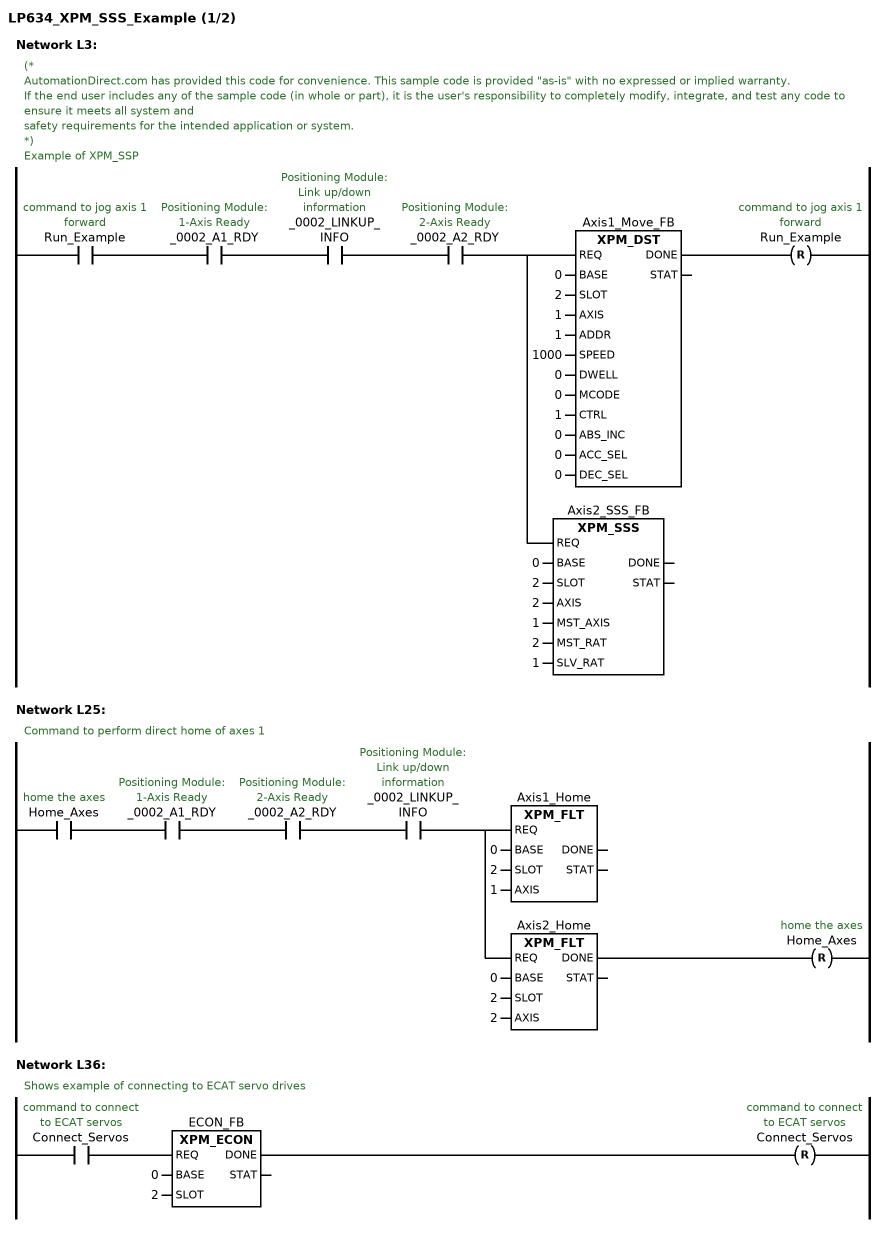
(* [picture p48: LP634_XPM_SSS_Example rungs L3-L36] *)
(* ( * / AutomationDirect.com has provided this code for convenience. This sample code is provided "as-is" with no expressed or implied warranty. / If the end user includes any of the sample code (in whole or part), it is the user's responsibility to completely modify, integrate, and test any code to ensure it meets all system and / safety requirements for the intended application or system. / * ) *)
(* Example of XPM_SSP *)
(* Rung L3 *)
_p1 := Run_Example AND _0002_A1_RDY AND _0002_LINKUP_INFO AND _0002_A2_RDY;
Axis1_Move_FB(REQ := _p1, BASE := 0, SLOT := 2, AXIS := 1, ADDR := 1, SPEED := 1000, DWELL := 0, MCODE := 0, CTRL := 1, ABS_INC := 0, ACC_SEL := 0, DEC_SEL := 0);
IF Axis1_Move_FB.DONE THEN Run_Example := FALSE; END_IF;
Axis2_SSS_FB(REQ := _p1, BASE := 0, SLOT := 2, AXIS := 2, MST_AXIS := 1, MST_RAT := 2, SLV_RAT := 1);
(* Command to perform direct home of axes 1 *)
(* Rung L25 *)
_p2 := Home_Axes AND _0002_A1_RDY AND _0002_A2_RDY AND _0002_LINKUP_INFO;
Axis1_Home(REQ := _p2, BASE := 0, SLOT := 2, AXIS := 1);
Axis2_Home(REQ := _p2, BASE := 0, SLOT := 2, AXIS := 2);
IF Axis2_Home.DONE THEN Home_Axes := FALSE; END_IF;
(* Shows example of connecting to ECAT servo drives *)
(* Rung L36 *)
ECON_FB(REQ := Connect_Servos, BASE := 0, SLOT := 2);
IF ECON_FB.DONE THEN Connect_Servos := FALSE; END_IF;

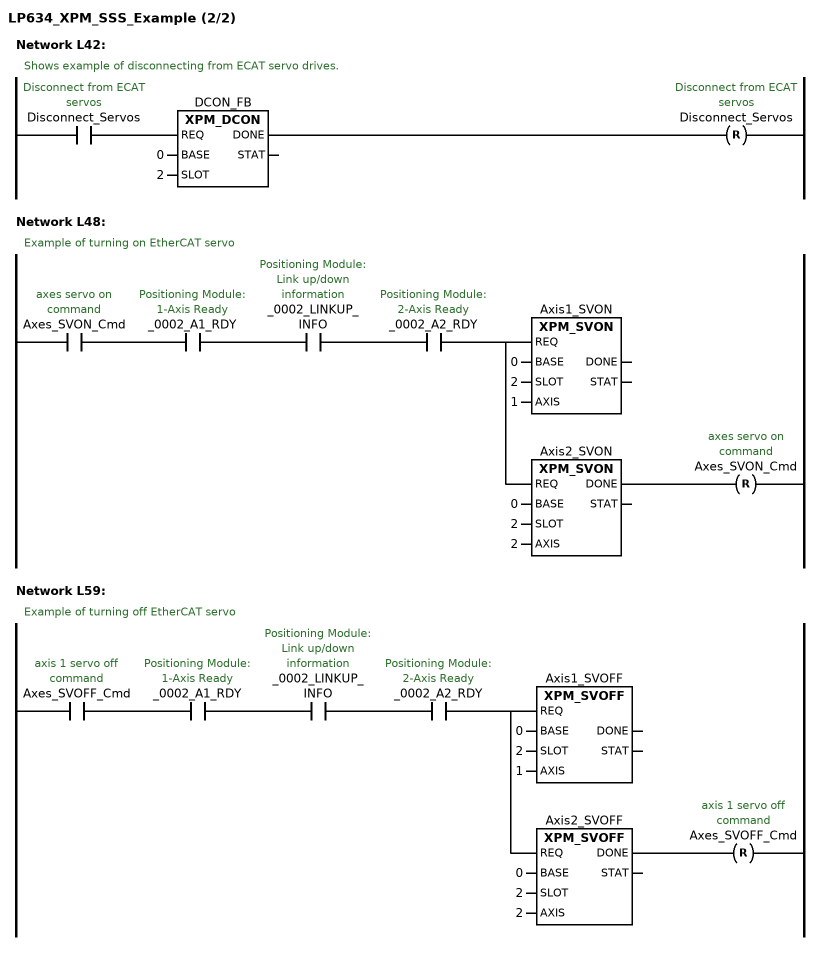
(* Shows example of disconnecting from ECAT servo drives. *)
(* Rung L42 *)
DCON_FB(REQ := Disconnect_Servos, BASE := 0, SLOT := 2);
IF DCON_FB.DONE THEN Disconnect_Servos := FALSE; END_IF;
(* Example of turning on EtherCAT servo *)
(* Rung L48 *)
_p3 := Axes_SVON_Cmd AND _0002_A1_RDY AND _0002_LINKUP_INFO AND _0002_A2_RDY;
Axis1_SVON(REQ := _p3, BASE := 0, SLOT := 2, AXIS := 1);
Axis2_SVON(REQ := _p3, BASE := 0, SLOT := 2, AXIS := 2);
IF Axis2_SVON.DONE THEN Axes_SVON_Cmd := FALSE; END_IF;
(* Example of turning off EtherCAT servo *)
(* Rung L59 *)
_p4 := Axes_SVOFF_Cmd AND _0002_A1_RDY AND _0002_LINKUP_INFO AND _0002_A2_RDY;
Axis1_SVOFF(REQ := _p4, BASE := 0, SLOT := 2, AXIS := 1);
Axis2_SVOFF(REQ := _p4, BASE := 0, SLOT := 2, AXIS := 2);
IF Axis2_SVOFF.DONE THEN Axes_SVOFF_Cmd := FALSE; END_IF;
END_PROGRAM

PROGRAM LP634_XPM_SSSP_Example (* task: Scan Program *)
(* example program for XPM_SSSP *)
VAR
    Axes_SVOFF_Cmd : BOOL; (* axis 1 servo off command *)
    Axes_SVON_Cmd : BOOL; (* axes servo on command *)
    Axis1_Home : XPM_FLT; (* direct home of axis 1 *)
    Axis1_Move_FB : XPM_DST; (* axis 1 speed move fb *)
    Axis1_SVOFF : XPM_SVOFF; (* function block for axis 1 servo off *)
    Axis1_SVON : XPM_SVON; (* SVON fb for axis 1 *)
    Axis2_Home : XPM_FLT; (* direct home of axis 1 *)
    Axis2_SSSP_FB : XPM_SSSP; (* axis 2 XPM_SSSP fb *)
    Axis2_SVOFF : XPM_SVOFF; (* function block for axis 1 servo off *)
    Axis2_SVON : XPM_SVON; (* SVON fb for axis 1 *)
    Connect_Servos : BOOL; (* command to connect to ECAT servos *)
    DCON_FB : XPM_DCON; (* EtherCAT disconnect FB *)
    Disconnect_Servos : BOOL; (* Disconnect from ECAT servos *)
    ECON_FB : XPM_ECON; (* EtherCAT connect FB *)
    Home_Axes : BOOL; (* home the axes *)
    Run_Example : BOOL; (* command to jog axis 1 forward *)
END_VAR
VAR_EXTERNAL
    _0002_A1_RDY : BOOL; (* AT %UX0.2.0 *) (* Positioning Module: 1-Axis Ready *)
    _0002_A2_RDY : BOOL; (* AT %UX0.2.1 *) (* Positioning Module: 2-Axis Ready *)
    _0002_LINKUP_INFO : BOOL; (* AT %UX0.2.14 *) (* Positioning Module: Link up/down information *)
END_VAR
VAR
    _p1 : BOOL;
    _p2 : BOOL;
    _p3 : BOOL;
    _p4 : BOOL;
END_VAR

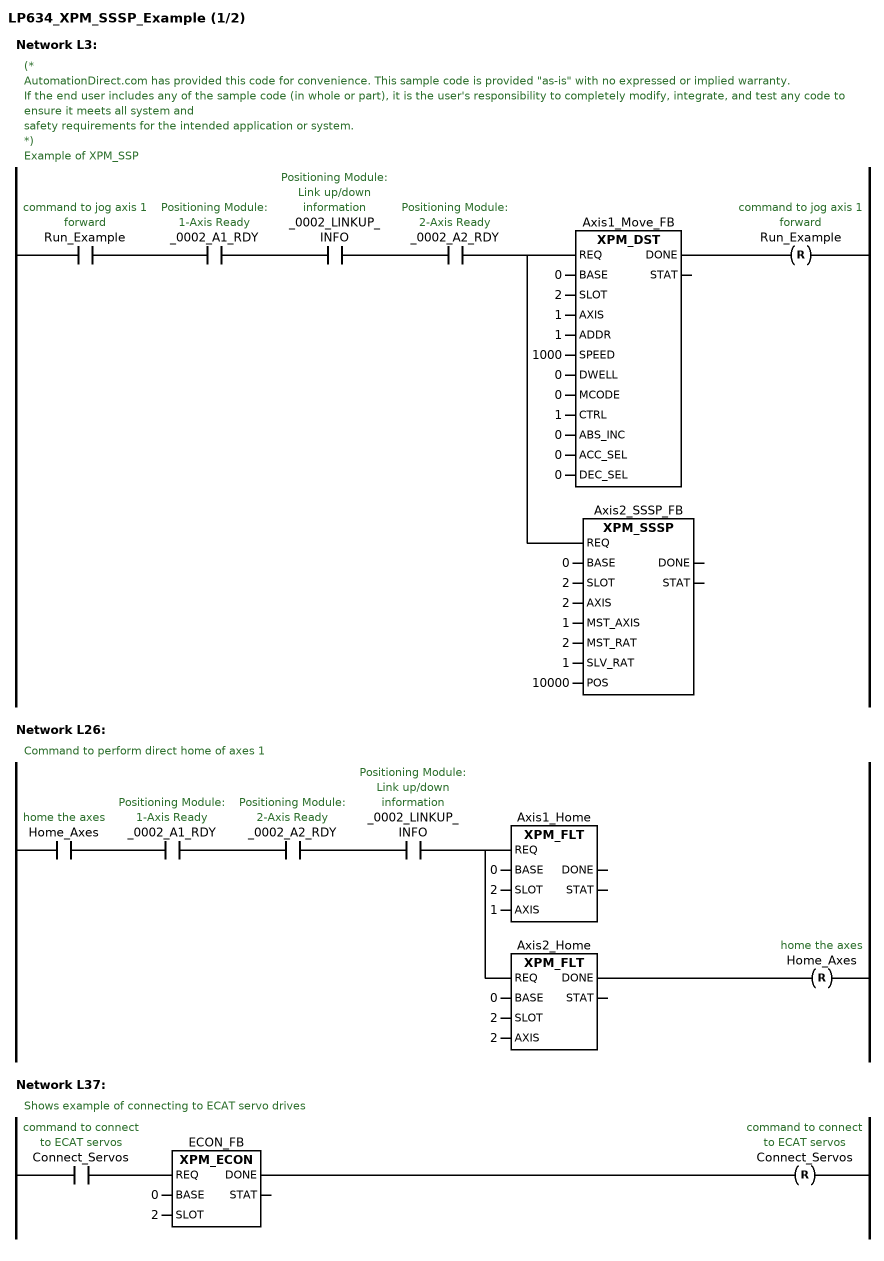
(* ( * / AutomationDirect.com has provided this code for convenience. This sample code is provided "as-is" with no expressed or implied warranty. / If the end user includes any of the sample code (in whole or part), it is the user's responsibility to completely modify, integrate, and test any code to ensure it meets all system and / safety requirements for the intended application or system. / * ) *)
(* Example of XPM_SSP *)
(* Rung L3 *)
_p1 := Run_Example AND _0002_A1_RDY AND _0002_LINKUP_INFO AND _0002_A2_RDY;
Axis1_Move_FB(REQ := _p1, BASE := 0, SLOT := 2, AXIS := 1, ADDR := 1, SPEED := 1000, DWELL := 0, MCODE := 0, CTRL := 1, ABS_INC := 0, ACC_SEL := 0, DEC_SEL := 0);
IF Axis1_Move_FB.DONE THEN Run_Example := FALSE; END_IF;
Axis2_SSSP_FB(REQ := _p1, BASE := 0, SLOT := 2, AXIS := 2, MST_AXIS := 1, MST_RAT := 2, SLV_RAT := 1, POS := 10000);
(* Command to perform direct home of axes 1 *)
(* Rung L26 *)
_p2 := Home_Axes AND _0002_A1_RDY AND _0002_A2_RDY AND _0002_LINKUP_INFO;
Axis1_Home(REQ := _p2, BASE := 0, SLOT := 2, AXIS := 1);
Axis2_Home(REQ := _p2, BASE := 0, SLOT := 2, AXIS := 2);
IF Axis2_Home.DONE THEN Home_Axes := FALSE; END_IF;
(* Shows example of connecting to ECAT servo drives *)
(* Rung L37 *)
ECON_FB(REQ := Connect_Servos, BASE := 0, SLOT := 2);
IF ECON_FB.DONE THEN Connect_Servos := FALSE; END_IF;

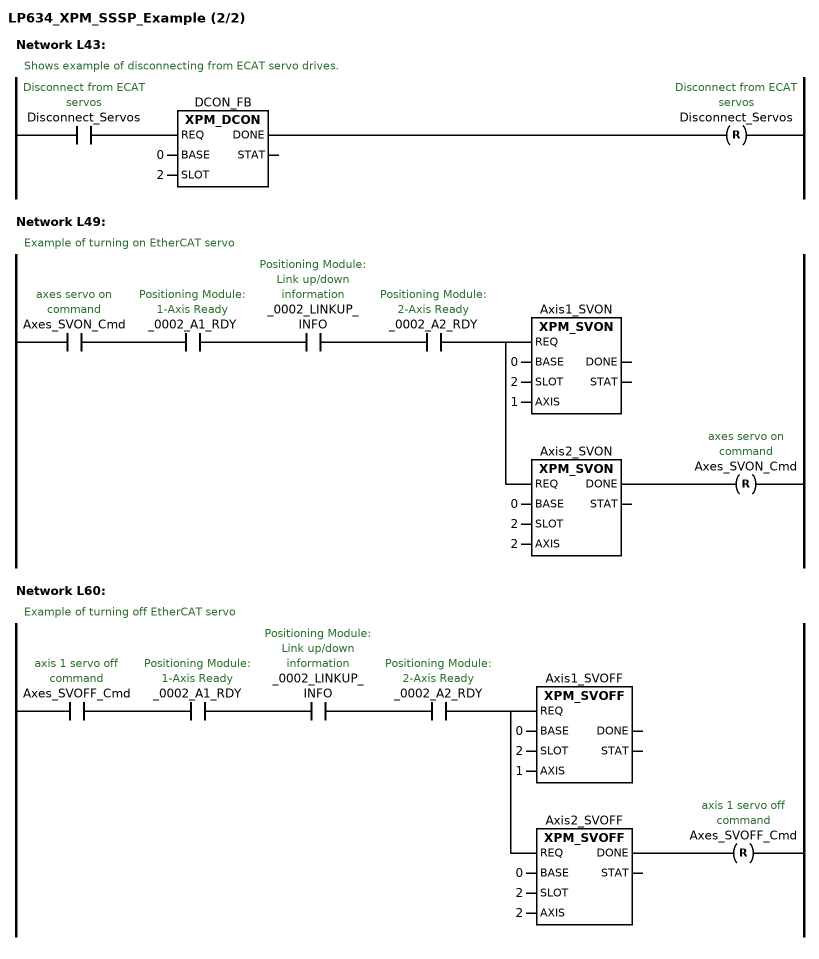
(* Shows example of disconnecting from ECAT servo drives. *)
(* Rung L43 *)
DCON_FB(REQ := Disconnect_Servos, BASE := 0, SLOT := 2);
IF DCON_FB.DONE THEN Disconnect_Servos := FALSE; END_IF;
(* Example of turning on EtherCAT servo *)
(* Rung L49 *)
_p3 := Axes_SVON_Cmd AND _0002_A1_RDY AND _0002_LINKUP_INFO AND _0002_A2_RDY;
Axis1_SVON(REQ := _p3, BASE := 0, SLOT := 2, AXIS := 1);
Axis2_SVON(REQ := _p3, BASE := 0, SLOT := 2, AXIS := 2);
IF Axis2_SVON.DONE THEN Axes_SVON_Cmd := FALSE; END_IF;
(* Example of turning off EtherCAT servo *)
(* Rung L60 *)
_p4 := Axes_SVOFF_Cmd AND _0002_A1_RDY AND _0002_LINKUP_INFO AND _0002_A2_RDY;
Axis1_SVOFF(REQ := _p4, BASE := 0, SLOT := 2, AXIS := 1);
Axis2_SVOFF(REQ := _p4, BASE := 0, SLOT := 2, AXIS := 2);
IF Axis2_SVOFF.DONE THEN Axes_SVOFF_Cmd := FALSE; END_IF;
END_PROGRAM

PROGRAM LP635_XPM_ELIN_Example (* task: Scan Program *)
(* example program for XPM_ELIN  function block. *)
VAR
    Axes_SVOFF_Cmd : BOOL; (* axis 1 servo off command *)
    Axes_SVON_Cmd : BOOL; (* axes servo on command *)
    Axis1_CMD_Step : UINT; (* step to run in XPM_IST *)
    Axis1_ELIN : XPM_ELIN; (* xpm ELIN fb *)
    Axis1_ELIN_CMD : BOOL; (* command to jog axis 1 forward *)
    Axis1_Home : XPM_FLT; (* direct home of axis 1 *)
    Axis1_SVOFF : XPM_SVOFF; (* function block for axis 1 servo off *)
    Axis1_SVON : XPM_SVON; (* SVON fb for axis 1 *)
    Axis2_Home : XPM_FLT; (* direct home of axis 1 *)
    Axis2_SVOFF : XPM_SVOFF; (* function block for axis 1 servo off *)
    Axis2_SVON : XPM_SVON; (* SVON fb for axis 1 *)
    Connect_Servos : BOOL; (* command to connect to ECAT servos *)
    DCON_FB : XPM_DCON; (* EtherCAT disconnect FB *)
    Disconnect_Servos : BOOL; (* Disconnect from ECAT servos *)
    ECON_FB : XPM_ECON; (* EtherCAT connect FB *)
    Home_Axes : BOOL; (* home the axes *)
END_VAR
VAR_EXTERNAL
    _0002_A1_RDY : BOOL; (* AT %UX0.2.0 *) (* Positioning Module: 1-Axis Ready *)
    _0002_A2_RDY : BOOL; (* AT %UX0.2.1 *) (* Positioning Module: 2-Axis Ready *)
    _0002_LINKUP_INFO : BOOL; (* AT %UX0.2.14 *) (* Positioning Module: Link up/down information *)
END_VAR
VAR
    _p1 : BOOL;
    _p2 : BOOL;
    _p3 : BOOL;
END_VAR

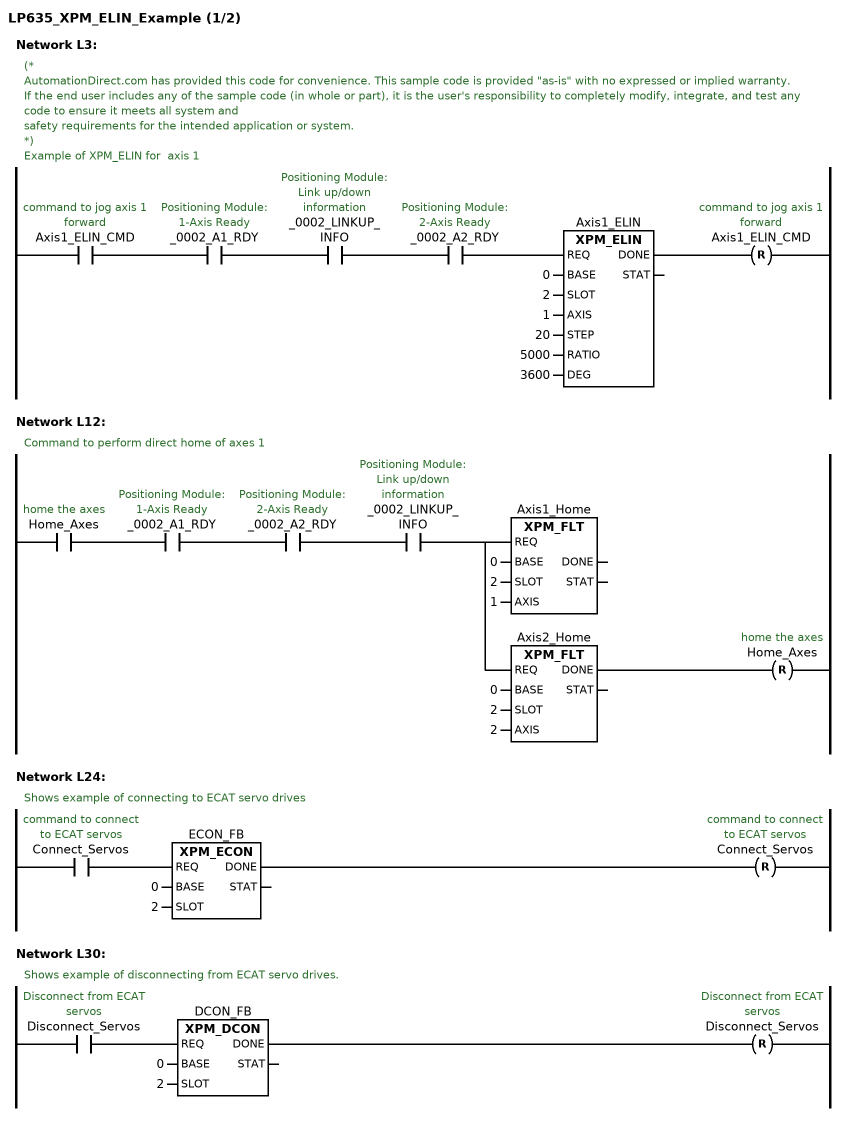
(* ( * / AutomationDirect.com has provided this code for convenience. This sample code is provided "as-is" with no expressed or implied warranty. / If the end user includes any of the sample code (in whole or part), it is the user's responsibility to completely modify, integrate, and test any code to ensure it meets all system and / safety requirements for the intended application or system. / * ) *)
(* Example of XPM_ELIN for  axis 1 *)
(* Rung L3 *)
Axis1_ELIN(REQ := Axis1_ELIN_CMD AND _0002_A1_RDY AND _0002_LINKUP_INFO AND _0002_A2_RDY, BASE := 0, SLOT := 2, AXIS := 1, STEP := 20, RATIO := 5000, DEG := 3600);
IF Axis1_ELIN.DONE THEN Axis1_ELIN_CMD := FALSE; END_IF;
(* Command to perform direct home of axes 1 *)
(* Rung L12 *)
_p1 := Home_Axes AND _0002_A1_RDY AND _0002_A2_RDY AND _0002_LINKUP_INFO;
Axis1_Home(REQ := _p1, BASE := 0, SLOT := 2, AXIS := 1);
Axis2_Home(REQ := _p1, BASE := 0, SLOT := 2, AXIS := 2);
IF Axis2_Home.DONE THEN Home_Axes := FALSE; END_IF;
(* Shows example of connecting to ECAT servo drives *)
(* Rung L24 *)
ECON_FB(REQ := Connect_Servos, BASE := 0, SLOT := 2);
IF ECON_FB.DONE THEN Connect_Servos := FALSE; END_IF;
(* Shows example of disconnecting from ECAT servo drives. *)
(* Rung L30 *)
DCON_FB(REQ := Disconnect_Servos, BASE := 0, SLOT := 2);
IF DCON_FB.DONE THEN Disconnect_Servos := FALSE; END_IF;

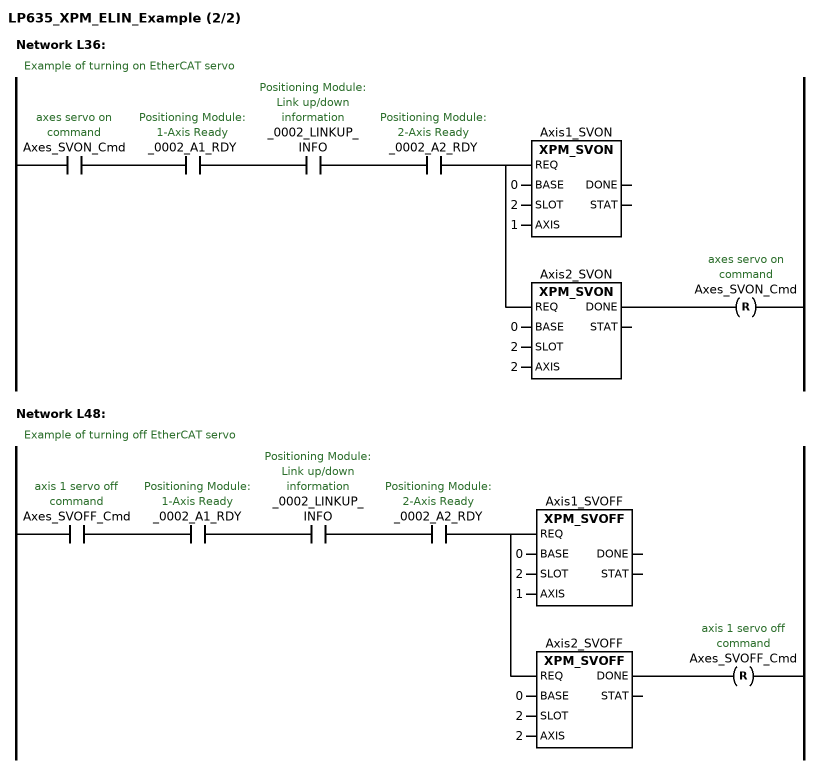
(* Example of turning on EtherCAT servo *)
(* Rung L36 *)
_p2 := Axes_SVON_Cmd AND _0002_A1_RDY AND _0002_LINKUP_INFO AND _0002_A2_RDY;
Axis1_SVON(REQ := _p2, BASE := 0, SLOT := 2, AXIS := 1);
Axis2_SVON(REQ := _p2, BASE := 0, SLOT := 2, AXIS := 2);
IF Axis2_SVON.DONE THEN Axes_SVON_Cmd := FALSE; END_IF;
(* Example of turning off EtherCAT servo *)
(* Rung L48 *)
_p3 := Axes_SVOFF_Cmd AND _0002_A1_RDY AND _0002_LINKUP_INFO AND _0002_A2_RDY;
Axis1_SVOFF(REQ := _p3, BASE := 0, SLOT := 2, AXIS := 1);
Axis2_SVOFF(REQ := _p3, BASE := 0, SLOT := 2, AXIS := 2);
IF Axis2_SVOFF.DONE THEN Axes_SVOFF_Cmd := FALSE; END_IF;
END_PROGRAM

PROGRAM LP636_XPM_CAM_Example (* task: Scan Program *)
(* example program for XPM_CAM *)
VAR
    Axes_SVOFF_Cmd : BOOL; (* axis 1 servo off command *)
    Axes_SVON_Cmd : BOOL; (* axes servo on command *)
    Axis1_Home : XPM_FLT; (* direct home of axis 1 *)
    Axis1_Move_FB : XPM_DST; (* axis 1 speed move fb *)
    Axis1_SVOFF : XPM_SVOFF; (* function block for axis 1 servo off *)
    Axis1_SVON : XPM_SVON; (* SVON fb for axis 1 *)
    Axis2_CAM_FB : XPM_CAM; (* axis 2 XPM_CAM fb *)
    Axis2_Home : XPM_FLT; (* direct home of axis 1 *)
    Axis2_SVOFF : XPM_SVOFF; (* function block for axis 1 servo off *)
    Axis2_SVON : XPM_SVON; (* SVON fb for axis 1 *)
    Connect_Servos : BOOL; (* command to connect to ECAT servos *)
    DCON_FB : XPM_DCON; (* EtherCAT disconnect FB *)
    Disconnect_Servos : BOOL; (* Disconnect from ECAT servos *)
    ECON_FB : XPM_ECON; (* EtherCAT connect FB *)
    Home_Axes : BOOL; (* home the axes *)
    Run_Example : BOOL; (* command to jog axis 1 forward *)
END_VAR
VAR_EXTERNAL
    _0002_A1_RDY : BOOL; (* AT %UX0.2.0 *) (* Positioning Module: 1-Axis Ready *)
    _0002_A2_RDY : BOOL; (* AT %UX0.2.1 *) (* Positioning Module: 2-Axis Ready *)
    _0002_LINKUP_INFO : BOOL; (* AT %UX0.2.14 *) (* Positioning Module: Link up/down information *)
END_VAR
VAR
    _p1 : BOOL;
    _p2 : BOOL;
    _p3 : BOOL;
    _p4 : BOOL;
END_VAR

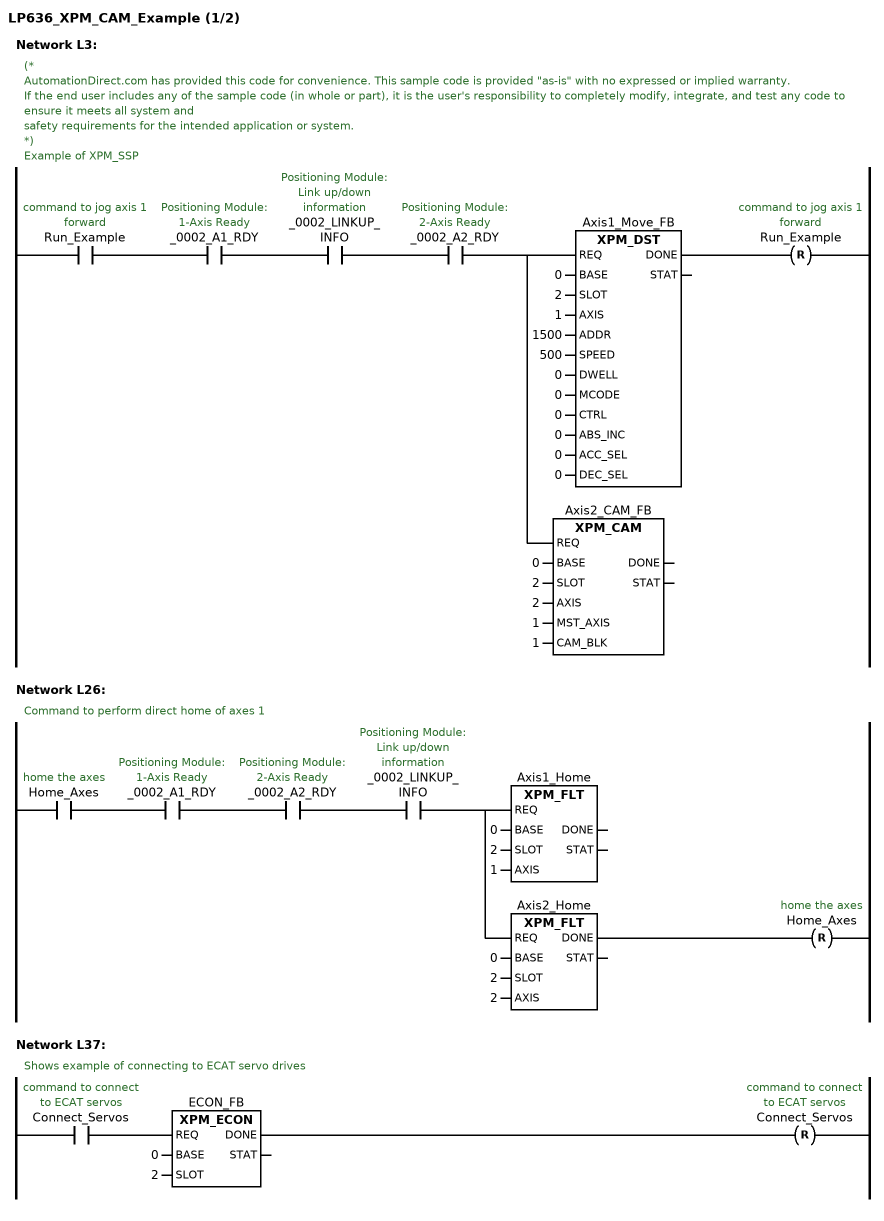
(* ( * / AutomationDirect.com has provided this code for convenience. This sample code is provided "as-is" with no expressed or implied warranty. / If the end user includes any of the sample code (in whole or part), it is the user's responsibility to completely modify, integrate, and test any code to ensure it meets all system and / safety requirements for the intended application or system. / * ) *)
(* Example of XPM_SSP *)
(* Rung L3 *)
_p1 := Run_Example AND _0002_A1_RDY AND _0002_LINKUP_INFO AND _0002_A2_RDY;
Axis1_Move_FB(REQ := _p1, BASE := 0, SLOT := 2, AXIS := 1, ADDR := 1500, SPEED := 500, DWELL := 0, MCODE := 0, CTRL := 0, ABS_INC := 0, ACC_SEL := 0, DEC_SEL := 0);
IF Axis1_Move_FB.DONE THEN Run_Example := FALSE; END_IF;
Axis2_CAM_FB(REQ := _p1, BASE := 0, SLOT := 2, AXIS := 2, MST_AXIS := 1, CAM_BLK := 1);
(* Command to perform direct home of axes 1 *)
(* Rung L26 *)
_p2 := Home_Axes AND _0002_A1_RDY AND _0002_A2_RDY AND _0002_LINKUP_INFO;
Axis1_Home(REQ := _p2, BASE := 0, SLOT := 2, AXIS := 1);
Axis2_Home(REQ := _p2, BASE := 0, SLOT := 2, AXIS := 2);
IF Axis2_Home.DONE THEN Home_Axes := FALSE; END_IF;
(* Shows example of connecting to ECAT servo drives *)
(* Rung L37 *)
ECON_FB(REQ := Connect_Servos, BASE := 0, SLOT := 2);
IF ECON_FB.DONE THEN Connect_Servos := FALSE; END_IF;

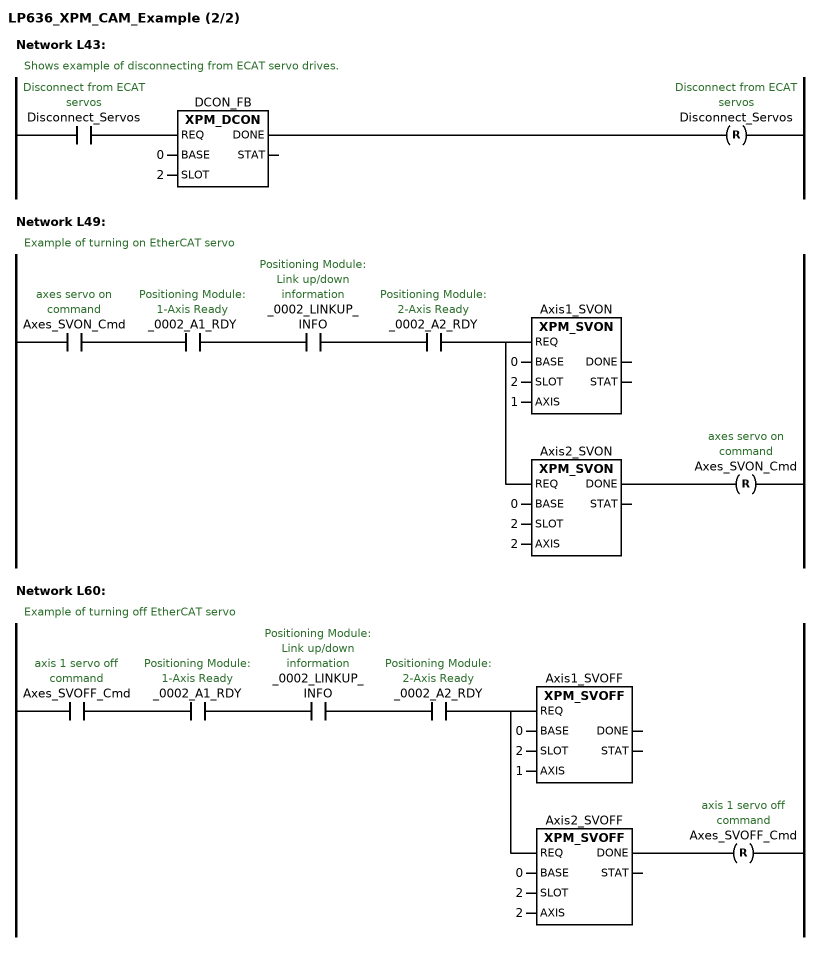
(* Shows example of disconnecting from ECAT servo drives. *)
(* Rung L43 *)
DCON_FB(REQ := Disconnect_Servos, BASE := 0, SLOT := 2);
IF DCON_FB.DONE THEN Disconnect_Servos := FALSE; END_IF;
(* Example of turning on EtherCAT servo *)
(* Rung L49 *)
_p3 := Axes_SVON_Cmd AND _0002_A1_RDY AND _0002_LINKUP_INFO AND _0002_A2_RDY;
Axis1_SVON(REQ := _p3, BASE := 0, SLOT := 2, AXIS := 1);
Axis2_SVON(REQ := _p3, BASE := 0, SLOT := 2, AXIS := 2);
IF Axis2_SVON.DONE THEN Axes_SVON_Cmd := FALSE; END_IF;
(* Example of turning off EtherCAT servo *)
(* Rung L60 *)
_p4 := Axes_SVOFF_Cmd AND _0002_A1_RDY AND _0002_LINKUP_INFO AND _0002_A2_RDY;
Axis1_SVOFF(REQ := _p4, BASE := 0, SLOT := 2, AXIS := 1);
Axis2_SVOFF(REQ := _p4, BASE := 0, SLOT := 2, AXIS := 2);
IF Axis2_SVOFF.DONE THEN Axes_SVOFF_Cmd := FALSE; END_IF;
END_PROGRAM

PROGRAM LP636_XPM_CAMO_Example (* task: Scan Program *)
(* example program for XPM_CAMO *)
VAR
    Axes_SVOFF_Cmd : BOOL; (* axis 1 servo off command *)
    Axes_SVON_Cmd : BOOL; (* axes servo on command *)
    Axis1_Home : XPM_FLT; (* direct home of axis 1 *)
    Axis1_Move_FB : XPM_DST; (* axis 1 speed move fb *)
    Axis1_SVOFF : XPM_SVOFF; (* function block for axis 1 servo off *)
    Axis1_SVON : XPM_SVON; (* SVON fb for axis 1 *)
    Axis2_CAMO_FB : XPM_CAMO; (* axis 2 XPM_CAMO fb *)
    Axis2_Home : XPM_FLT; (* direct home of axis 1 *)
    Axis2_SVOFF : XPM_SVOFF; (* function block for axis 1 servo off *)
    Axis2_SVON : XPM_SVON; (* SVON fb for axis 1 *)
    Connect_Servos : BOOL; (* command to connect to ECAT servos *)
    DCON_FB : XPM_DCON; (* EtherCAT disconnect FB *)
    Disconnect_Servos : BOOL; (* Disconnect from ECAT servos *)
    ECON_FB : XPM_ECON; (* EtherCAT connect FB *)
    Home_Axes : BOOL; (* home the axes *)
    Run_Example : BOOL; (* command to jog axis 1 forward *)
END_VAR
VAR_EXTERNAL
    _0002_A1_RDY : BOOL; (* AT %UX0.2.0 *) (* Positioning Module: 1-Axis Ready *)
    _0002_A2_RDY : BOOL; (* AT %UX0.2.1 *) (* Positioning Module: 2-Axis Ready *)
    _0002_LINKUP_INFO : BOOL; (* AT %UX0.2.14 *) (* Positioning Module: Link up/down information *)
END_VAR
VAR
    _p1 : BOOL;
    _p2 : BOOL;
    _p3 : BOOL;
    _p4 : BOOL;
END_VAR

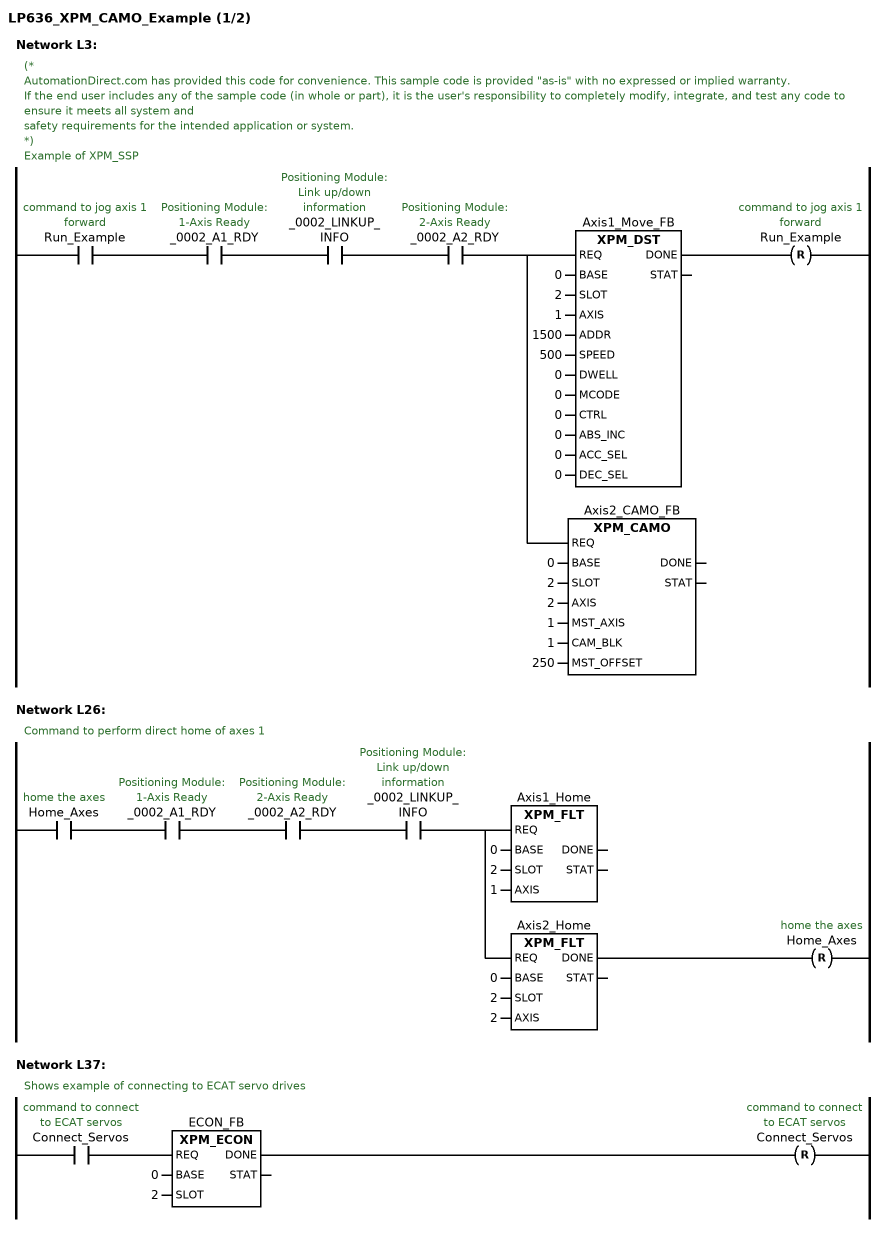
(* ( * / AutomationDirect.com has provided this code for convenience. This sample code is provided "as-is" with no expressed or implied warranty. / If the end user includes any of the sample code (in whole or part), it is the user's responsibility to completely modify, integrate, and test any code to ensure it meets all system and / safety requirements for the intended application or system. / * ) *)
(* Example of XPM_SSP *)
(* Rung L3 *)
_p1 := Run_Example AND _0002_A1_RDY AND _0002_LINKUP_INFO AND _0002_A2_RDY;
Axis1_Move_FB(REQ := _p1, BASE := 0, SLOT := 2, AXIS := 1, ADDR := 1500, SPEED := 500, DWELL := 0, MCODE := 0, CTRL := 0, ABS_INC := 0, ACC_SEL := 0, DEC_SEL := 0);
IF Axis1_Move_FB.DONE THEN Run_Example := FALSE; END_IF;
Axis2_CAMO_FB(REQ := _p1, BASE := 0, SLOT := 2, AXIS := 2, MST_AXIS := 1, CAM_BLK := 1, MST_OFFSET := 250);
(* Command to perform direct home of axes 1 *)
(* Rung L26 *)
_p2 := Home_Axes AND _0002_A1_RDY AND _0002_A2_RDY AND _0002_LINKUP_INFO;
Axis1_Home(REQ := _p2, BASE := 0, SLOT := 2, AXIS := 1);
Axis2_Home(REQ := _p2, BASE := 0, SLOT := 2, AXIS := 2);
IF Axis2_Home.DONE THEN Home_Axes := FALSE; END_IF;
(* Shows example of connecting to ECAT servo drives *)
(* Rung L37 *)
ECON_FB(REQ := Connect_Servos, BASE := 0, SLOT := 2);
IF ECON_FB.DONE THEN Connect_Servos := FALSE; END_IF;

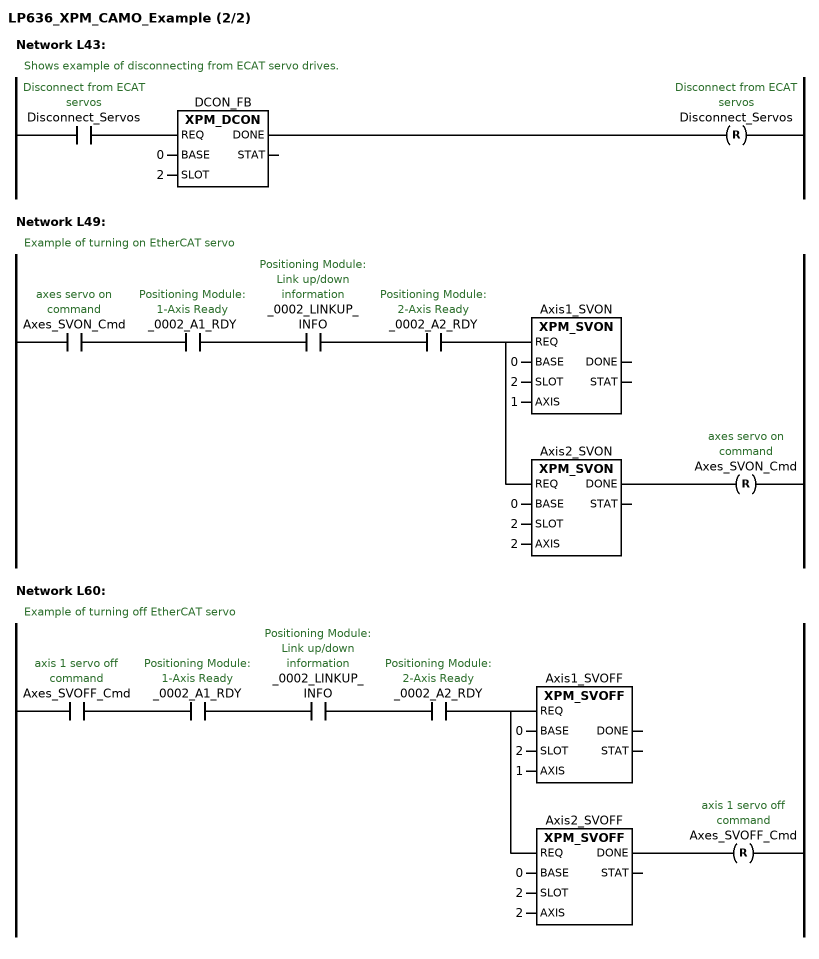
(* Shows example of disconnecting from ECAT servo drives. *)
(* Rung L43 *)
DCON_FB(REQ := Disconnect_Servos, BASE := 0, SLOT := 2);
IF DCON_FB.DONE THEN Disconnect_Servos := FALSE; END_IF;
(* Example of turning on EtherCAT servo *)
(* Rung L49 *)
_p3 := Axes_SVON_Cmd AND _0002_A1_RDY AND _0002_LINKUP_INFO AND _0002_A2_RDY;
Axis1_SVON(REQ := _p3, BASE := 0, SLOT := 2, AXIS := 1);
Axis2_SVON(REQ := _p3, BASE := 0, SLOT := 2, AXIS := 2);
IF Axis2_SVON.DONE THEN Axes_SVON_Cmd := FALSE; END_IF;
(* Example of turning off EtherCAT servo *)
(* Rung L60 *)
_p4 := Axes_SVOFF_Cmd AND _0002_A1_RDY AND _0002_LINKUP_INFO AND _0002_A2_RDY;
Axis1_SVOFF(REQ := _p4, BASE := 0, SLOT := 2, AXIS := 1);
Axis2_SVOFF(REQ := _p4, BASE := 0, SLOT := 2, AXIS := 2);
IF Axis2_SVOFF.DONE THEN Axes_SVOFF_Cmd := FALSE; END_IF;
END_PROGRAM